FUNCTION_BLOCK BOOLTEST (* Test Boolean AND,OR,XOR *)
  (* Standard: 61131-3 *)
  (* Version 0.0, 2004-12-15, JHC, Rockwell Automation, Converted from SRC format. *)
  (* Compiler header: package fb.rt.plc.bits; *)
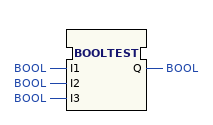
  VAR_INPUT
    I1 : BOOL;
    I2 : BOOL;
    I3 : BOOL;
  END_VAR
  VAR_OUTPUT
    Q : BOOL;
  END_VAR
  ALGORITHM REQ IN FBD:
    FBS
      n1 : NOT_BOOL;
      n2 : NOT_BOOL;
      a1 : AND_BOOL;
      a2 : AND_BOOL;
      o1 : OR_BOOL;
      x1 : XOR_BOOL;
    END_FBS
    DATA_CONNECTIONS
      I1 TO n1.in;
      I2 TO n2.in;
      I2 TO a1.i2;
      n2.Q TO a2.i2;
      n1.Q TO a1.i1;
      I1 TO a2.i1;
      a1.Q TO o1.i1;
      a2.Q TO o1.i2;
      o1.Q TO x1.i1;
      I3 TO x1.i2;
      x1.Q TO Q;
    END_CONNECTIONS
  END_ALGORITHM
END_FUNCTION_BLOCK
